Yaskawa INFORM job: kufsa_new.JBI

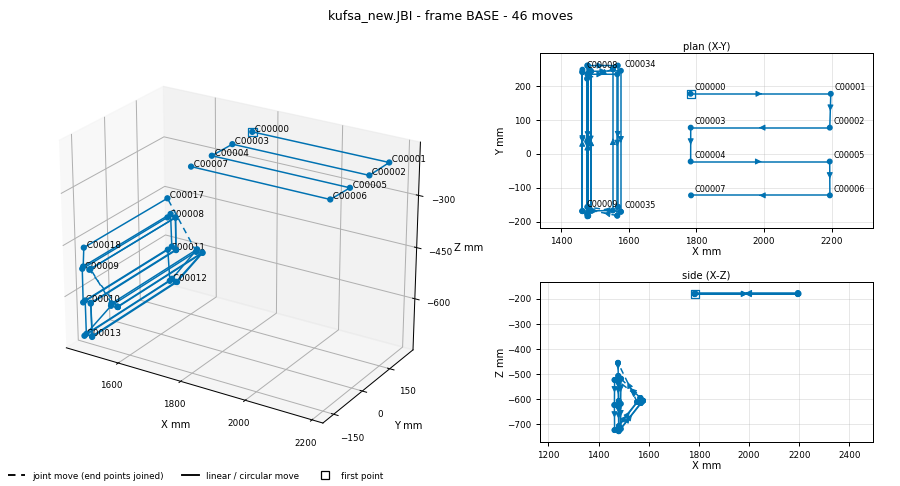
[picture p0: tool path of kufsa_new.JBI in frame BASE, 46 of 51 moves have a stored position in this frame; points joined in program order, loops and branches not executed]
/JOB
//NAME kufsa_new
//POS
///NPOS 46,0,46,0,0,0
///TOOL 0
///POSTYPE BASE
///RECTAN
///RCONF 0,0,0,0,0,0,0,0,0,0,0,0,0,0,0,0,0,0,0,0,0,0,0,0
C00000=1783.333279,177.683675,-178.952236,175.000000,5.000000,90.000000
C00001=2197.437272,177.683675,-178.952236,175.000000,5.000000,90.000000
C00002=2194.402886,77.683675,-180.929062,175.000000,5.000000,90.000000
C00003=1783.689385,77.683675,-180.929062,175.000000,5.000000,90.000000
C00004=1783.507651,-22.316325,-180.005624,175.000000,5.000000,90.000000
C00005=2194.164298,-22.316325,-180.005624,175.000000,5.000000,90.000000
C00006=2194.697568,-122.316325,-175.996333,175.000000,5.000000,90.000000
C00007=1784.686125,-122.316325,-175.996333,175.000000,5.000000,90.000000
C00008=1464.014944,241.444919,-522.722824,175.000000,-89.999999,5.000000
C00009=1464.014944,-169.159182,-522.722824,175.000000,-89.999999,5.000000
C00010=1463.152146,-168.687677,-622.722824,175.000000,-89.999999,5.000000
C00011=1463.152146,242.022110,-622.722824,175.000000,-89.999999,5.000000
C00012=1463.935741,248.955843,-722.722824,175.000000,-89.999999,5.000000
C00013=1463.935741,-168.695364,-722.722824,175.000000,-89.999999,5.000000
C00014=1553.861020,-166.978204,-610.590790,180.000000,-45.000000,0.000000
C00015=1553.861020,250.441215,-610.590790,180.000000,-45.000000,0.000000
C00016=1553.861020,250.441215,-610.590790,180.000000,-45.000000,0.000000
C00017=1477.531479,222.423079,-454.518710,175.000000,-89.999999,5.000000
C00018=1477.531479,-177.571334,-454.518710,175.000000,-89.999999,5.000000
C00019=1478.554227,-184.306124,-506.723051,175.000000,-89.999999,5.000000
C00020=1478.554227,235.762831,-506.723051,175.000000,-89.999999,5.000000
C00021=1480.684642,236.380115,-606.723051,175.000000,-89.999999,5.000000
C00022=1480.684642,-183.074602,-606.723051,175.000000,-89.999999,5.000000
C00023=1480.955307,-182.919266,-706.723051,175.000000,-89.999999,5.000000
C00024=1480.955307,235.380836,-706.723051,175.000000,-89.999999,5.000000
C00025=1566.683394,235.369668,-594.591017,180.000000,-45.000000,0.000000
C00026=1566.683394,-182.153753,-594.591017,180.000000,-45.000000,0.000000
C00027=1566.683394,-182.153753,-594.591017,180.000000,-45.000000,0.000000
C00028=1489.401467,-166.687872,-517.941327,175.000000,-89.999999,5.000000
C00029=1489.401467,243.705577,-517.941327,175.000000,-89.999999,5.000000
C00030=1488.117436,245.937237,-617.941327,175.000000,-89.999999,5.000000
C00031=1488.117436,-168.048822,-617.941327,175.000000,-89.999999,5.000000
C00032=1488.292841,-166.510367,-717.941327,175.000000,-89.999999,5.000000
C00033=1488.292841,243.987327,-717.941327,175.000000,-89.999999,5.000000
C00034=1577.392093,245.653806,-605.809293,180.000000,-45.000000,0.000000
C00035=1577.392093,-170.654707,-605.809293,180.000000,-45.000000,0.000000
C00036=1577.392093,-170.654707,-605.809293,180.000000,-45.000000,0.000000
C00037=1478.179092,-156.595710,-527.111793,175.000000,-89.999999,5.000000
C00038=1478.179092,261.165284,-527.111793,175.000000,-89.999999,5.000000
C00039=1479.297370,260.284031,-627.111793,175.000000,-89.999999,5.000000
C00040=1479.297370,-156.550276,-627.111793,175.000000,-89.999999,5.000000
C00041=1480.372619,-156.285545,-727.111793,175.000000,-89.999999,5.000000
C00042=1480.372619,260.999795,-727.111793,175.000000,-89.999999,5.000000
C00043=1568.328511,261.113252,-614.979759,180.000000,-45.000000,0.000000
C00044=1568.328511,-156.025890,-614.979759,180.000000,-45.000000,0.000000
C00045=1568.328511,-156.025890,-614.979759,180.000000,-45.000000,0.000000
///POSTYPE PULSE
///PULSE
EC00000=0
EC00001=0
EC00002=0
EC00003=0
EC00004=0
EC00005=0
EC00006=0
EC00007=0
EC00008=0
EC00009=0
EC00010=0
EC00011=0
EC00012=0
EC00013=0
EC00014=0
EC00015=0
EC00016=92160
EC00017=92160
EC00018=92160
EC00019=92160
EC00020=92160
EC00021=92160
EC00022=92160
EC00023=92160
EC00024=92160
EC00025=92160
EC00026=92160
EC00027=184320
EC00028=184320
EC00029=184320
EC00030=184320
EC00031=184320
EC00032=184320
EC00033=184320
EC00034=184320
EC00035=184320
EC00036=276480
EC00037=276480
EC00038=276480
EC00039=276480
EC00040=276480
EC00041=276480
EC00042=276480
EC00043=276480
EC00044=276480
EC00045=368640
//INST
///DATE 2023/01/19 10:50
///ATTR SC,RW,RJ
////FRAME BASE
///GROUP1 RB1,ST1
NOP
MOVJ C00000 EC00000 VJ=15.0
CALL JOB:SPYON
MOVL C00001 EC00001 V=200.0
MOVL C00002 EC00002 V=200.0
MOVL C00003 EC00003 V=200.0
MOVL C00004 EC00004 V=200.0
MOVL C00005 EC00005 V=200.0
MOVL C00006 EC00006 V=200.0
MOVL C00007 EC00007 V=200.0
CALL JOB:SPYOF
MOVJ P009 VJ=15.00
MOVJ C00008 EC00008 VJ=15.0
CALL JOB:SPYON
MOVL C00009 EC00009 V=200.0
MOVL C00010 EC00010 V=200.0
MOVL C00011 EC00011 V=200.0
MOVL C00012 EC00012 V=200.0
MOVL C00013 EC00013 V=200.0
MOVL C00014 EC00014 V=200.0
MOVL C00015 EC00015 V=200.0
CALL JOB:SPYOF
MOVJ P009 VJ=15.00
MOVL C00016 EC00016 V=200.0
MOVJ C00017 EC00017 VJ=15.0
CALL JOB:SPYON
MOVL C00018 EC00018 V=200.0
MOVL C00019 EC00019 V=200.0
MOVL C00020 EC00020 V=200.0
MOVL C00021 EC00021 V=200.0
MOVL C00022 EC00022 V=200.0
MOVL C00023 EC00023 V=200.0
MOVL C00024 EC00024 V=200.0
MOVL C00025 EC00025 V=200.0
MOVL C00026 EC00026 V=200.0
CALL JOB:SPYOF
MOVJ P009 VJ=15.00
MOVL C00027 EC00027 V=200.0
MOVJ C00028 EC00028 VJ=15.0
CALL JOB:SPYON
MOVL C00029 EC00029 V=200.0
MOVL C00030 EC00030 V=200.0
MOVL C00031 EC00031 V=200.0
MOVL C00032 EC00032 V=200.0
MOVL C00033 EC00033 V=200.0
MOVL C00034 EC00034 V=200.0
MOVL C00035 EC00035 V=200.0
CALL JOB:SPYOF
MOVJ P009 VJ=15.00
MOVL C00036 EC00036 V=200.0
MOVJ C00037 EC00037 VJ=15.0
CALL JOB:SPYON
MOVL C00038 EC00038 V=200.0
MOVL C00039 EC00039 V=200.0
MOVL C00040 EC00040 V=200.0
MOVL C00041 EC00041 V=200.0
MOVL C00042 EC00042 V=200.0
MOVL C00043 EC00043 V=200.0
MOVL C00044 EC00044 V=200.0
CALL JOB:SPYOF
MOVJ P009 VJ=15.00
MOVL C00045 EC00045 V=200.0
END
